KUKA KRL program: HG_EKRL.src, HG_EKRL.dat

--- HG_EKRL.src ---
&ACCESS RVO1
&REL 257
&PARAM EDITMASK = *
&PARAM TEMPLATE = C:\KRC\Roboter\Template\vorgabe
&PARAM DISKPATH = KRC:\R1\Program\KRL
DEF HG_EKRL( )
;fold DECL
DECL INT TTTT
DECL CHAR Bytes[32]
DECL EKI_STATUS RET
;endfold
;FOLD INI;%{PE}
  ;FOLD BASISTECH INI
    GLOBAL INTERRUPT DECL 3 WHEN $STOPMESS==TRUE DO IR_STOPM ( )
    INTERRUPT ON 3
    BAS (#INITMOV,0 )
  ;ENDFOLD (BASISTECH INI)
  ;FOLD USER INI
    ;Make your modifications here

  ;ENDFOLD (USER INI)

;ENDFOLD (INI)
;------------



EKRL_CONNECT()



;Bytes[]="hellow"
;halt

;EKRL_Close()
END

GLOBAL DEF EKRL_Vision_Int_Data(EKRL_NAME:IN)
DECL CHAR Message_Error[1024],EKRL_NAME[]
DECL EKI_STATUS RET
DECL  BOOL IsStatus
Message_Error[]=" "
IsStatus=false

EKRL_Connect(EKRL_NAME[])


RET=EKI_SetString(EKRL_NAME[],"KUKA_Receive/@Model","Vision_Ini_Data")
RET = EKI_Send(EKRL_NAME[],"KUKA_Receive")


Message_Wait("Wait Vision Int Data!",2)


RET=EKI_GetBool(EKRL_NAME[],"KUKA_Send/@IsStatus" ,IsStatus)
RET=EKI_GetString(EKRL_NAME[],"KUKA_Send/Message_Error" ,Message_Error[])
RET=EKI_GetINT(EKRL_NAME[],"KUKA_Send/Initialization_Data/Vision_Scope" ,Vision_Scope)


RET=EKI_Close(EKRL_NAME[])
RET=EKI_Clear(EKRL_NAME[])

IF  IsStatus THEN

MSGNOTIFY(Message_Error[])

else

MsgQuit(Message_Error[], "HanGao")
halt
ENDIF


END

GLOBAL DEF EKRL_Find_Model_Send(EKRL_NAME:IN,Work_Number:IN,Find_Area:IN)
DECL INT ID,Work,Find_Area,OPFFSET,Work_Number,Find_Data_Model
DECL CHAR Find_Area_String[1024], Message_Error[1024],Message_Show[1024],Work_Area[1024],EKRL_NAME[]
DECL BOOL Calculation_Status
DECL Frame LastPos1,LastPos2,LastPos3,LastPos4,LastPos5,LastPos6,LastPos7,LastPos8,LastPos9
DECL E6POS LP1,LP2,LP3,LP4,LP5,LP6,LP7,LP8,LP9

DECL EKI_STATUS RET
DECL State_t _State,STAT
DECL MODUS_T MODE
MODE=#SYNC



OPFFSET=0
Calculation_Status=false
$Flag[2]=false
LastPos1={X 0.0,Y 0.0,A 0.0,B 0.0,C 0.0}
LastPos2={X 0.0,Y 0.0,A 0.0,B 0.0,C 0.0}
LastPos3={X 0.0,Y 0.0,A 0.0,B 0.0,C 0.0}
LastPos4={X 0.0,Y 0.0,A 0.0,B 0.0,C 0.0}
LastPos5={X 0.0,Y 0.0,A 0.0,B 0.0,C 0.0}
LastPos6={X 0.0,Y 0.0,A 0.0,B 0.0,C 0.0}
LastPos7={X 0.0,Y 0.0,A 0.0,B 0.0,C 0.0}
LastPos8={X 0.0,Y 0.0,A 0.0,B 0.0,C 0.0}
LastPos9={X 0.0,Y 0.0,A 0.0,B 0.0,C 0.0}
LP1={X 0.0,Y 0.0,A 0.0,B 0.0,C 0.0}
LP2={X 0.0,Y 0.0,A 0.0,B 0.0,C 0.0}
LP3={X 0.0,Y 0.0,A 0.0,B 0.0,C 0.0}
LP4={X 0.0,Y 0.0,A 0.0,B 0.0,C 0.0}
LP5={X 0.0,Y 0.0,A 0.0,B 0.0,C 0.0}
LP6={X 0.0,Y 0.0,A 0.0,B 0.0,C 0.0}
LP7={X 0.0,Y 0.0,A 0.0,B 0.0,C 0.0}
LP8={X 0.0,Y 0.0,A 0.0,B 0.0,C 0.0}
LP9={X 0.0,Y 0.0,A 0.0,B 0.0,C 0.0}


Find_Area_String[]=" "
Message_Error[]=" "
Message_Show[]=" "



EKRL_Connect(EKRL_NAME[])


switch Find_Area

CASE 1

Find_Area_String[]="F_45"

CASE 2
Find_Area_String[]="F_135"

CASE 3
Find_Area_String[]="F_225"

CASE 4
Find_Area_String[]="F_315"

ENDSWITCH


switch Work_Number

CASE 1

Work_Area[]="Work_1"

Find_Data_Model=N1_Sink_Data.Sink_Model


CASE 2
Work_Area[]="Work_2"
Find_Data_Model=N2_Sink_Data.Sink_Model
CASE 3
Work_Area[]="Work_3"

CASE 4
Work_Area[]="Work_4"

ENDSWITCH

RET=EKI_SetString(EKRL_NAME[],"KUKA_Receive/@Model","Find_Model")
RET=EKI_SetInt(EKRL_NAME[],"KUKA_Receive/Find_Model/@Find_Data", Find_Data_Model)
RET=EKI_SetString(EKRL_NAME[],"KUKA_Receive/Find_Model/@Work_Area", Work_Area[])
RET=EKI_SetString(EKRL_NAME[],"KUKA_Receive/Find_Model/@Vision_Area", Find_Area_String[])
RET=EKI_SetFrame(EKRL_NAME[],"KUKA_Receive/Camera_Point/Pos_1", $POS_ACT)

RET = EKI_Send(EKRL_NAME[],"KUKA_Receive")


Message_Wait("Find Model Data Sending",2)

RET=EKI_GetBool(EKRL_NAME[],"KUKA_Send/@IsStatus" ,Calculation_Status)
RET=EKI_GetString(EKRL_NAME[],"KUKA_Send/Message_Error" ,Message_Error[])

SWRITE( Message_Show[] , _State , OPFFSET ,"Vision Find Model: %s"  ,Message_Error[] )
IF  Calculation_Status THEN


RET=EKI_GetFrame(EKRL_NAME[],"KUKA_Send/Vision_Point/Pos_1" ,LastPos1)
RET=EKI_GetFrame(EKRL_NAME[],"KUKA_Send/Vision_Point/Pos_2" ,LastPos2)
RET=EKI_GetFrame(EKRL_NAME[],"KUKA_Send/Vision_Point/Pos_3" ,LastPos3)
RET=EKI_GetFrame(EKRL_NAME[],"KUKA_Send/Vision_Point/Pos_4" ,LastPos4)
RET=EKI_GetFrame(EKRL_NAME[],"KUKA_Send/Vision_Point/Pos_5" ,LastPos5)
RET=EKI_GetFrame(EKRL_NAME[],"KUKA_Send/Vision_Point/Pos_6" ,LastPos6)
RET=EKI_GetFrame(EKRL_NAME[],"KUKA_Send/Vision_Point/Pos_7" ,LastPos7)
RET=EKI_GetFrame(EKRL_NAME[],"KUKA_Send/Vision_Point/Pos_8" ,LastPos8)
RET=EKI_GetFrame(EKRL_NAME[],"KUKA_Send/Vision_Point/Pos_9" ,LastPos9)
LP1=LastPos1
LP2=LastPos2
LP3=LastPos3
LP4=LastPos4
LP5=LastPos5
LP6=LastPos6
LP7=LastPos7
LP8=LastPos8
LP9=LastPos9


HanGao_Camera_Offset(#Find_Model ,Find_Area,Work_Number,LP1)
HanGao_Camera_Offset(#Find_Model ,Find_Area,Work_Number,LP2)
HanGao_Camera_Offset(#Find_Model ,Find_Area,Work_Number,LP3)
HanGao_Camera_Offset(#Find_Model ,Find_Area,Work_Number,LP4)

switch Find_Area

CASE 1

N45_OFFSET_POS=LP2
N45_CIR_POS=LP1
D45_Start_POS=LP4
D45_End_POS=LP3
CASE 2
N135_OFFSET_POS=LP2
N135_CIR_POS=LP1
D135_Start_POS=LP4
D135_End_POS=LP3
CASE 3
N225_OFFSET_POS=LP2
N225_CIR_POS=LP1
D225_Start_POS=LP4
D225_End_POS=LP3
CASE 4
N315_OFFSET_POS=LP2
N315_CIR_POS=LP1
D315_Start_POS=LP4
D315_End_POS=LP3
ENDSWITCH


MSGNOTIFY(Message_Error[],"HanGao")
else



MsgQuit(Message_Error[], "HanGao")
halt
;return


ENDIF


RET=EKI_Close(EKRL_NAME[])
RET=EKI_Clear(EKRL_NAME[])

End


GLOBAL DEF  Message_Wait(Msg_String:IN,Flag_No:IN)
DECL CHAR Msg_String[]
DECL INT Flag_No
DECL INT Mess_INT
DECL BOOL Mess_Del
Mess_INT=-1

REPEAT
;halt
IF NOT Exists_KrlMsg(Mess_INT) THEN
Msg_Wait(Msg_String[],false,Mess_INT,Flag_No)
;halt
ENDIF


UNTIL  $Flag[Flag_No]
Mess_Del=Clear_KrlMsg(Mess_INT)


END



GLOBAL DEF EKRL_Calibration_Send(EKRL_NAME:IN,Area_Name:IN,Work_Area:IN)
DECL INT Area_Name,Calibration_Mark,Work_Area
DECL CHAR Message_Error[1024],Work_Area_Name[1024],EKRL_NAME[]
DECL EKI_STATUS RET
DECL BOOL Calibration_Status
DECL Frame LastPos1,LastPos2,LastPos3,LastPos4,LastPos5,LastPos6,LastPos7,LastPos8,LastPos9
;-----INI--------
$Flag[2]=FALSE
Calibration_Status=False
$Flag[2]=false
Message_Error[]=" "
Work_Area_Name[]=" "
LastPos1={X 0.0,Y 0.0,A 0.0,B 0.0,C 0.0}
LastPos2={X 0.0,Y 0.0,A 0.0,B 0.0,C 0.0}
LastPos3={X 0.0,Y 0.0,A 0.0,B 0.0,C 0.0}
LastPos4={X 0.0,Y 0.0,A 0.0,B 0.0,C 0.0}
LastPos5={X 0.0,Y 0.0,A 0.0,B 0.0,C 0.0}
LastPos6={X 0.0,Y 0.0,A 0.0,B 0.0,C 0.0}
LastPos7={X 0.0,Y 0.0,A 0.0,B 0.0,C 0.0}
LastPos8={X 0.0,Y 0.0,A 0.0,B 0.0,C 0.0}
LastPos9={X 0.0,Y 0.0,A 0.0,B 0.0,C 0.0}
;-----INI--------

EKRL_Connect(EKRL_NAME[])


switch Work_Area

CASE 1

Work_Area_Name[]="Work_1"

Calibration_Mark=N1_Sink_Data.Sink_Model

CASE 2
Work_Area_Name[]="Work_2"
Calibration_Mark=N2_Sink_Data.Sink_Model
CASE 3
Work_Area_Name[]="Work_3"

CASE 4
Work_Area_Name[]="Work_4"

ENDSWITCH


SWITCH Area_Name

CASE 1
RET=EKI_SetString(EKRL_NAME[],"KUKA_Receive/Calibration_Model/@Vision_Area","F_45")

switch Work_Area
CASE 1
RET=EKI_SetFrame(EKRL_NAME[],"KUKA_Receive/Camera_Point/Pos_1", N1_Cam_45_POS)

CASE 2
RET=EKI_SetFrame(EKRL_NAME[],"KUKA_Receive/Camera_Point/Pos_1", N2_Cam_45_POS)
CASE 3

CASE 4
ENDSWITCH


CASE 2
RET=EKI_SetString(EKRL_NAME[],"KUKA_Receive/Calibration_Model/@Vision_Area","F_135")
switch Work_Area
CASE 1
RET=EKI_SetFrame(EKRL_NAME[],"KUKA_Receive/Camera_Point/Pos_1", N1_Cam_135_POS)

CASE 2
RET=EKI_SetFrame(EKRL_NAME[],"KUKA_Receive/Camera_Point/Pos_1", N2_Cam_135_POS)
CASE 3

CASE 4
ENDSWITCH

CASE 3
RET=EKI_SetString(EKRL_NAME[],"KUKA_Receive/Calibration_Model/@Vision_Area","F_225")
switch Work_Area
CASE 1
RET=EKI_SetFrame(EKRL_NAME[],"KUKA_Receive/Camera_Point/Pos_1", N1_Cam_225_POS)

CASE 2
RET=EKI_SetFrame(EKRL_NAME[],"KUKA_Receive/Camera_Point/Pos_1", N2_Cam_225_POS)
CASE 3

CASE 4
ENDSWITCH
CASE 4
RET=EKI_SetString(EKRL_NAME[],"KUKA_Receive/Calibration_Model/@Vision_Area","F_315")
switch Work_Area
CASE 1
RET=EKI_SetFrame(EKRL_NAME[],"KUKA_Receive/Camera_Point/Pos_1", N1_Cam_315_POS)

CASE 2
RET=EKI_SetFrame(EKRL_NAME[],"KUKA_Receive/Camera_Point/Pos_1", N2_Cam_315_POS)
CASE 3

CASE 4
ENDSWITCH
ENDSWITCH


switch	Global_Calib_Model


case #New

RET=EKI_SetFrame(EKRL_NAME[],"KUKA_Receive/Vision_Point/Pos_1", Calibration_Point[1])
RET=EKI_SetFrame(EKRL_NAME[],"KUKA_Receive/Vision_Point/Pos_2", Calibration_Point[2])
RET=EKI_SetFrame(EKRL_NAME[],"KUKA_Receive/Vision_Point/Pos_3", Calibration_Point[3])
RET=EKI_SetFrame(EKRL_NAME[],"KUKA_Receive/Vision_Point/Pos_4", Calibration_Point[4])
RET=EKI_SetFrame(EKRL_NAME[],"KUKA_Receive/Vision_Point/Pos_5", Calibration_Point[5])
RET=EKI_SetFrame(EKRL_NAME[],"KUKA_Receive/Vision_Point/Pos_6", Calibration_Point[6])
RET=EKI_SetFrame(EKRL_NAME[],"KUKA_Receive/Vision_Point/Pos_7", Calibration_Point[7])
RET=EKI_SetFrame(EKRL_NAME[],"KUKA_Receive/Vision_Point/Pos_8", Calibration_Point[8])
RET=EKI_SetFrame(EKRL_NAME[],"KUKA_Receive/Vision_Point/Pos_9", Calibration_Point[9])

RET=EKI_SetString(EKRL_NAME[],"KUKA_Receive/@Model","Calibration_New")


case #Add

RET=EKI_SetString(EKRL_NAME[],"KUKA_Receive/@Model","Calibration_Add")

case #Text

RET=EKI_SetString(EKRL_NAME[],"KUKA_Receive/@Model","Calibration_Text")




endSwitch



RET=EKI_SetString(EKRL_NAME[],"KUKA_Receive/Calibration_Model/@Work_Area", Work_Area_Name[])
RET=EKI_SetInt(EKRL_NAME[],"KUKA_Receive/Calibration_Model/@Calibration_Mark", Calibration_Mark)



RET = EKI_Send(EKRL_NAME[],"KUKA_Receive")



Message_Wait("Calibration Data Sending",2)



RET=EKI_GetBool(EKRL_NAME[],"KUKA_Send/@IsStatus" ,Calibration_Status)
RET=EKI_GetString(EKRL_NAME[],"KUKA_Send/Message_Error" ,Message_Error[])


IF  Calibration_Status THEN

switch Global_Calib_Model

case #Text


RET=EKI_GetFrame(EKRL_NAME[],"KUKA_Send/Vision_Point/Pos_1" ,LastPos1)
RET=EKI_GetFrame(EKRL_NAME[],"KUKA_Send/Vision_Point/Pos_2" ,LastPos2)
RET=EKI_GetFrame(EKRL_NAME[],"KUKA_Send/Vision_Point/Pos_3" ,LastPos3)
RET=EKI_GetFrame(EKRL_NAME[],"KUKA_Send/Vision_Point/Pos_4" ,LastPos4)
RET=EKI_GetFrame(EKRL_NAME[],"KUKA_Send/Vision_Point/Pos_5" ,LastPos5)
RET=EKI_GetFrame(EKRL_NAME[],"KUKA_Send/Vision_Point/Pos_6" ,LastPos6)
RET=EKI_GetFrame(EKRL_NAME[],"KUKA_Send/Vision_Point/Pos_7" ,LastPos7)
RET=EKI_GetFrame(EKRL_NAME[],"KUKA_Send/Vision_Point/Pos_8" ,LastPos8)
RET=EKI_GetFrame(EKRL_NAME[],"KUKA_Send/Vision_Point/Pos_9" ,LastPos9)
Calibration_Text[1]=LastPos1
Calibration_Text[2]=LastPos2
Calibration_Text[3]=LastPos3
Calibration_Text[4]=LastPos4
Calibration_Text[5]=LastPos5
Calibration_Text[6]=LastPos6
Calibration_Text[7]=LastPos7
Calibration_Text[8]=LastPos8
Calibration_Text[9]=LastPos9
case #Add



endSwitch




MSGNOTIFY(Message_Error[])

else

MsgQuit(Message_Error[], "HanGao")
halt
ENDIF


RET=EKI_Close(EKRL_NAME[])
RET=EKI_Clear(EKRL_NAME[])
;wait until data read
;WAIT FOR $FLAG[1]



End



GLOBAL DEF EKRL_Connect(EKRL_NAME:IN)
DECL EKI_STATUS RET
DECL INT Mess_INT
DECL BOOL Mess_Del
DECL CHAR EKRL_NAME[]
;EKRL_NAME[]="HanGaoEkrl"
Mess_INT=-1
RET=EKI_Init(EKRL_NAME[])
EKI_CHECK(RET,#Quit,EKRL_NAME[])

;HALT
RET=EKI_OPEN(EKRL_NAME[])
EKI_CHECK(RET,#Quit,EKRL_NAME[])

wait sec 0.2

;MSGNOTIFY("HanGao:Socket Connecting!")


REPEAT
;halt
IF NOT Exists_KrlMsg(Mess_INT) THEN
Msg_Wait("Socket Connecting",false,Mess_INT,Connect_Falg)
;halt
ENDIF
IF NOT $FLAG[Connect_Falg]  THEN
RET=EKI_open(EKRL_NAME[])
;HALT

wait sec 2



ENDIF

UNTIL  $Flag[Connect_Falg]
Mess_Del=Clear_KrlMsg(Mess_INT)
MSGNOTIFY("HanGao:Socket Connecting OK!")


End
GLOBAL DEF EKRL_Close(EKRL_NAME:IN)
DECL CHAR EKRL_NAME[]
DECL EKI_STATUS RET
RET=EKI_Close(EKRL_NAME[])
RET=EKI_Clear(EKRL_NAME[])

END



GLOBAL  DEF  Msg_Wait(mess[]:IN,Wait_ON:IN,MSG_INT:OUT,Connect_Flag:IN)
DECL INT Msg_INT,Connect_Flag
DECL BOOL Msg_Clear,Msg_Exit,Wait_ON
DECL CHAR mess[]
DECL KRLMSG_T MYMESSAGE
DECL KRLMSGPAR_T Parameter[3]
DECL KRLMSGOPT_T Option
Msg_INT=-1
Msg_Clear=false
Msg_Exit=false
mymessage.Msg_txt[]=mess[]
MYMESSAGE.Modul[]="HanGao"
MYMESSAGE.Nr=1
Parameter[1]={Par_Type #EMPTY}
Parameter[2]={Par_Type #EMPTY}
Parameter[3]={Par_Type #EMPTY}
MSG_INT=SET_KRLMSG(#WAITING,MYMESSAGE,Parameter[],Option)

REPEAT
wait sec 0.012
IF $FLAG[Connect_Flag] THEN
Msg_Clear=Clear_KrlMsg(Msg_INT)
ENDIF
Msg_Exit=Exists_KrlMsg(Msg_INT)
UNTIL NOT(Msg_Exit) OR Msg_Clear OR NOT(WAIT_ON)
END

--- HG_EKRL.dat ---
&ACCESS RVO1
&REL 257
&PARAM EDITMASK = *
&PARAM TEMPLATE = C:\KRC\Roboter\Template\vorgabe
&PARAM DISKPATH = KRC:\R1\Program\KRL
DEFDAT  hg_ekrl PUBLIC


DECL INT SUCCESS



GLOBAL ENUM Find_Model_Enum F_45,F_135,F_225,F_315
GLOBAL ENUM Calib_Model_Enum New,Add,Text
DECL GLOBAL Calib_Model_Enum Global_Calib_Model=#Text

DECL GLOBAL INT Connect_Falg=1
DECL GLOBAL CHAR EKRL_NAME[1024]
DECL GLOBAL FRAME Calibration_Point[9]
Calibration_Point[1]={X 336.482086,Y 689.796,Z 1.13258839,A 0.284984082,B -0.0416393019,C -0.0681119189}
Calibration_Point[2]={X 334.470215,Y 656.540710,Z 1.13258791,A 0.284984052,B -0.0416393541,C -0.0681119040}
Calibration_Point[3]={X 332.504303,Y 622.809,Z 1.13258779,A 0.284984,B -0.0416393876,C -0.0681119}
Calibration_Point[4]={X 364.433960,Y 688.397217,Z 1.13260412,A 0.441926926,B -0.0416151658,C -0.0704161376}
Calibration_Point[5]={X 362.514709,Y 654.958923,Z 1.13260460,A 0.441926926,B -0.0416151248,C -0.0704161450}
Calibration_Point[6]={X 360.558197,Y 621.049,Z 1.13260412,A 0.441926867,B -0.0416151695,C -0.0704161227}
Calibration_Point[7]={X 392.662689,Y 686.764221,Z 1.19020331,A 0.441926807,B -0.0416152105,C -0.0704161078}
Calibration_Point[8]={X 390.848297,Y 653.285278,Z 1.13260353,A 0.441926748,B -0.0416152477,C -0.0704160929}
Calibration_Point[9]={X 388.725189,Y 619.578735,Z 1.13260090,A 0.441926926,B -0.0416151807,C -0.0704161301}

DECL GLOBAL FRAME Calibration_Text[9]
Calibration_Text[1]={X 336.541107,Y 689.730408,Z 0.0,A 0.0,B 0.0,C 0.0}
Calibration_Text[2]={X 334.499512,Y 656.518677,Z 0.0,A 0.0,B 0.0,C 0.0}
Calibration_Text[3]={X 332.507,Y 622.827698,Z 0.0,A 0.0,B 0.0,C 0.0}
Calibration_Text[4]={X 364.458,Y 688.385,Z 0.0,A 0.0,B 0.0,C 0.0}
Calibration_Text[5]={X 362.509399,Y 654.974609,Z 0.0,A 0.0,B 0.0,C 0.0}
Calibration_Text[6]={X 360.523499,Y 621.108398,Z 0.0,A 0.0,B 0.0,C 0.0}
Calibration_Text[7]={X 392.656,Y 686.779724,Z 0.0,A 0.0,B 0.0,C 0.0}
Calibration_Text[8]={X 390.811707,Y 653.345398,Z 0.0,A 0.0,B 0.0,C 0.0}
Calibration_Text[9]={X 388.842590,Y 619.442322,Z 0.0,A 0.0,B 0.0,C 0.0}

ENDDAT
